(* Copyright 2017 Cimpress

Licensed under the Apache License, Version 2.0 (the "License");
you may not use this file except in compliance with the License.
You may obtain a copy of the License at

http://www.apache.org/licenses/LICENSE-2.0

Unless required by applicable law or agreed to in writing, software
distributed under the License is distributed on an "AS IS" BASIS,
WITHOUT WARRANTIES OR CONDITIONS OF ANY KIND, either express or implied.
See the License for the specific language governing permissions and
limitations under the License. *)

TYPE T_Ctrl_AlarmConfig :
STRUCT
	// Disable the OFF Alarm transition
	bolOffAlarmTransitionDisable	: BOOL;
	// Disable the EOFF Alarm Transition
	bolEOffAlarmTransitionDisable	: BOOL;
	// Disable to Off Command Transition 
	bolOffCmdTransitionDisable		: BOOL;
	// Disable the EOffCommandTransition
	bolEOffCmdTransitionDisable		: BOOL;
	// Enable Alarm Propagation to Children
	bolChildrenAlarmPropagation		: BOOL;
END_STRUCT
END_TYPE

(* stored: Version 1.1.0.1, ProductVersion 3.1.4019.2
   DUT T_Ctrl_AlarmConfig: Id {aabd6e21-ed42-472e-a4fd-8e8bcbdc4f67} *)
